// TIA Portal V19 export
TYPE "C501_VAR_IF_KLH_TYPIC"
   STRUCT
      STS_OPEN { ExternalAccessible := 'False'; ExternalVisible := 'False'; ExternalWritable := 'False'} : Bool;   // Handbediende klep is open
      STS_TOE { ExternalAccessible := 'False'; ExternalVisible := 'False'; ExternalWritable := 'False'} : Bool;   // Handbediende klep is toe
      EXT_HW { ExternalAccessible := 'False'; ExternalVisible := 'False'; ExternalWritable := 'False'} : Bool;   // Sturings hardware (PLC) in storing
      STO { ExternalAccessible := 'False'; ExternalVisible := 'False'; ExternalWritable := 'False'} : Struct   // Opsomming van alle storingen
         A001 : Bool;   // Terugmeldingen Open en Dicht tegelijk
      END_STRUCT;
   END_STRUCT;
END_TYPE
